// TIA Portal V17 export
FUNCTION "FC_FanGasControl" : Void   // FC, LAD
{ S7_Optimized_Access := 'TRUE' }
   VAR_TEMP   // added for the SCL form of the ladder/FBD networks
      _variant1 : Variant;
      _real1 : Real;
   END_VAR
BEGIN

REGION Network 1: 风机输出
   // 风机运行控制和自动/手动模式选择输出
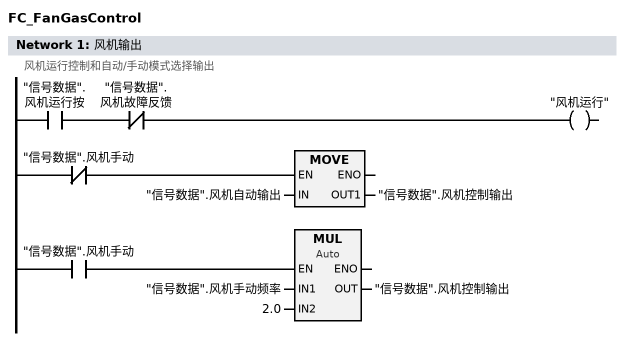
   RUNG wire#powerrail
      Contact( "信号数据".风机运行按 )
      I_Contact( "信号数据".风机故障反馈 )
      Coil( "风机运行" )
   END_RUNG
   RUNG wire#powerrail
      I_Contact( "信号数据".风机手动 )
      { S7_GenerateENO := "TRUE" } Move(in := "信号数据".风机自动输出, out1 => "信号数据".风机控制输出)
   END_RUNG
   RUNG wire#powerrail
      Contact( "信号数据".风机手动 )
      { S7_GenerateENO := "TRUE" } Mul(in1 := "信号数据".风机手动频率, in2 := 2.0, out => "信号数据".风机控制输出)
   END_RUNG
   // the same network as SCL:
   "风机运行" := "信号数据".风机运行按 AND NOT "信号数据".风机故障反馈;
   IF NOT "信号数据".风机手动 THEN "信号数据".风机控制输出 := "信号数据".风机自动输出; END_IF;
   IF "信号数据".风机手动 THEN "信号数据".风机控制输出 := "信号数据".风机手动频率 * 2.0; END_IF;
END_REGION

REGION Network 2: 风机输出计算
   // 停机清零、百分比换算和模拟量输出转换
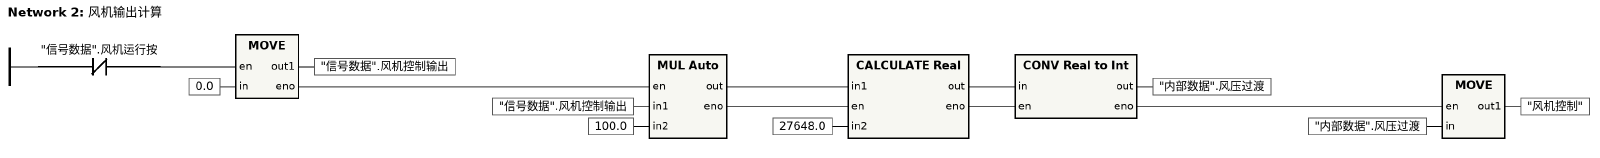
   RUNG wire#powerrail
      I_Contact( "信号数据".风机运行按 )
      { S7_GenerateENO := "TRUE" } Move(in := 0.0, out1 => "信号数据".风机控制输出)
      { S7_GenerateENO := "TRUE" } Mul(in1 := "信号数据".风机控制输出, in2 := 100.0, out => wire#w1)
      { S7_Templates := "SrcType := Real"; S7_GenerateENO := "TRUE"; S7_Expression := "IN1/IN2" } Calculate(in1 := wire#w2, in2 := 27648.0, out => wire#w3)
      { S7_Templates := "[SrcType := Real, DestType := Int]"; S7_GenerateENO := "TRUE" } Convert(in := wire#w4, out => "内部数据".风压过渡)
      { S7_GenerateENO := "TRUE" } Move(in := "内部数据".风压过渡, out1 => "风机控制")
   END_RUNG
   RUNG wire#w1
   END_RUNG wire#w2
   RUNG wire#w3
   END_RUNG wire#w4
   // the same network as SCL:
   // ENO of a box is taken as its EN; it also drops when the box reports an error
   IF NOT "信号数据".风机运行按 THEN
       "信号数据".风机控制输出 := 0.0;
       #_variant1 := "信号数据".风机控制输出 * 100.0;
       #_real1 := #_variant1/27648.0;
       "内部数据".风压过渡 := REAL_TO_INT(#_real1);
       "风机控制" := "内部数据".风压过渡;
   END_IF;
END_REGION

REGION Network 3: 燃气开启
   // 风压≥1.2时接通烧嘴电源
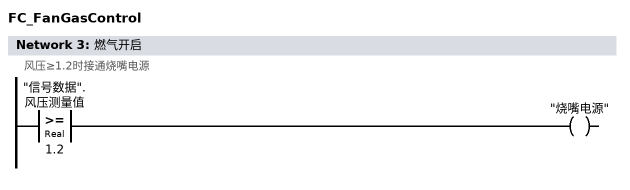
   RUNG wire#powerrail
      { S7_Templates := "SrcType := Real" } GE_Contact(in1 := "信号数据".风压测量值, in2 := 1.2)
      Coil( "烧嘴电源" )
   END_RUNG
   // the same network as SCL:
   "烧嘴电源" := "信号数据".风压测量值 >= 1.2;
END_REGION
END_FUNCTION
